VISUALIZATION NavBarEmpty  // 200x880
END_VISUALIZATION

(* stored: Version 1.1.0.1, ProductVersion 3.1.4024.9
   Visu NavBarEmpty: Id {99256d48-f1cf-45d6-9864-5f07d5a14b64} *)
